FUNCTION_BLOCK E_R_TRIG (* Composite Function Block Type *)
  (* Standard: 61499-2 *)
  (* Version 0.0, 9/9/2026, macie, Schneider Electric, template *)
  PACKAGE Main;
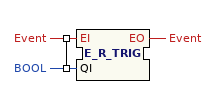
  EVENT_INPUT
    EI WITH QI; (* Initialization Request *)
  END_EVENT
  EVENT_OUTPUT
    EO; (* Initialization Confirm *)
  END_EVENT
  VAR_INPUT
    QI : BOOL := FALSE; (* Input event qualifier *)
  END_VAR
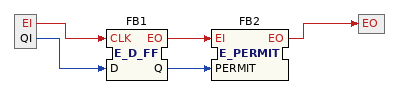
  FBS
    FB1 : E_D_FF;
    FB2 : E_PERMIT;
  END_FBS
  EVENT_CONNECTIONS
    FB2.EO TO EO;
    FB1.EO TO FB2.EI;
    EI TO FB1.CLK;
  END_CONNECTIONS
  DATA_CONNECTIONS
    QI TO FB1.D;
    FB1.Q TO FB2.PERMIT;
  END_CONNECTIONS
END_FUNCTION_BLOCK
